FUNCTION_BLOCK FB_PuckPicked
VAR_INPUT
	Execute : BOOL;
END_VAR
VAR_OUTPUT
	Done : BOOL;
END_VAR
VAR
	i: INT;
END_VAR

IF Execute THEN
	
	FOR i := 0 TO 38 DO
		memCpy(
			destAddr 	:= ADR(GVL.Pucks[i]),
			srcAddr 	:= ADR(GVL.Pucks[i+1]),
			n 			:= SIZEOF(GVL.Pucks[i+1])	
		);
	END_FOR

	IF GVL.puckIncrement < 1 THEN
		GVL.puckIncrement := GVL.puckIncrement;
	ELSE
		GVL.puckIncrement := GVL.puckIncrement - 1;
	END_IF
	Done := TRUE;
ELSE
	Done := FALSE;
END_IF

END_FUNCTION_BLOCK

(* stored: Version 1.1.0.1, ProductVersion 3.1.4024.11
   POU FB_PuckPicked: Id {a49f97a5-9545-4118-b081-f0deafa36c9c}, SpecialFunc None *)
